KUKA KRL data list: Folge125.dat

&ACCESS RVO1
&REL 5
&COMMENT Grundstellung
&PARAM DISKPATH = KRC:\R1\Folgen
&PARAM TEMPLATE = C:\KRC\Roboter\Template\vorgabe
&PARAM TPVW_VERSION = 8.1.8
&PARAM EDITMASK = Folge999[1-999]
DEFDAT FOLGE125
; interface to basic routines
EXT BAS (BAS_COMMAND :IN,REAL :IN )
; interface to VW-standard routines
EXT VW (VW_COMMAND:IN, BOOL: IN, REAL:IN, REAL:IN, REAL:IN, REAL:IN, BOOL :IN, E6POS :IN )
; interface to VW_USER - Call
EXT  VW_USER (VW_USER_CMD :IN,INT :IN,REAL  :IN,REAL  :IN,REAL  :IN,REAL  :IN,REAL  :IN,REAL  :IN,BOOL  :IN )
EXT  VW_USR_R (VW_USER_CMD :IN,INT :IN,REAL  :IN,REAL  :IN,REAL  :IN,REAL  :IN,REAL  :IN,REAL  :IN,BOOL  :IN )
EXT  IBGN (IBGN_COMMAND  :IN,BOOL  :IN,REAL  :IN,REAL  :IN,BOOL  :IN,E6POS  :OUT )
; interface select routine
EXTFCT INT  SELECT (SUBTYPE  :IN,INT  :IN,BOOL  :IN,ARI_TYP  :IN,INT  :IN,BOOL_TYP  :IN,INT  :IN,BOOL  :IN)
INT VW_NEXT_FREE = 2
INT VW_NFREE_SPS = 3
INT VW_MAX_SPS = 103
DECL VW_MPARA_TYP P0_D = {TOOL_NO 12,BASE_NO 0,VB 10,VE 0,ACC 100,TRG_TIME 0,MOVE_TYPE #PTP_MOTION}
DECL E6POS P0 = {X 1644.431, Y -174.7289, Z 2340.62, A 0.01137252, B 29.99963, C -90.35181, S 2, T 42 , E1 0.0, E2 0.0, E3 0.0, E4 0.0, E5 0.0, E6 0.0}
DECL VW_MPARA_TYP P1_D = {TOOL_NO 12,BASE_NO 0,VB 100,VE 0,ACC 100,TRG_TIME 0,MOVE_TYPE #PTP_MOTION}
DECL E6POS P1 = {X 1644.432, Y -174.729, Z 2340.621, A 0.01138396, B 29.99963, C -90.35179, S 2, T 42 , E1 0.0, E2 0.0, E3 0.0, E4 0.0, E5 0.0, E6 0.0}
ENDDAT
